{attribute 'linkalways'} 
{attribute 'no_explicit_call' := 'This FB is a CLASS and must be accessed using methods or properties'}
{attribute 'enable_dynamic_creation'}
FUNCTION_BLOCK _TcVnParamsMSER EXTENDS StructuredDatatypeBase
VAR
	localData : TcVnParamsMSER;
	activeData : REFERENCE TO TcVnParamsMSER REF= localData;
	_nDelta : _DINT(localData.nDelta);
    _nMinArea : _UDINT(localData.nMinArea);
	_nMaxArea : _UDINT(localData.nMaxArea);
	_fMaxVariation : _LREAL(localData.fMaxVariation);
	_fMinDiversity : _LREAL(localData.fMinDiversity);
	_nMaxEvolution : _UDINT(localData.nMaxEvolution);
    _fAreaThreshold : _LREAL(localData.fAreaThreshold);
    _fMinMargin : _LREAL(localData.fMinMargin);
    _nEdgeBlurSize : _UDINT(localData.nEdgeBlurSize);
END_VAR

PROPERTY PUBLIC Address : PVOID
GET
Address := ADR(activeData);
END_GET
END_PROPERTY

METHOD PUBLIC ClearReference
VAR_INPUT
END_VAR
activeData REF= localData;
SetMemberReference();
END_METHOD

METHOD PUBLIC Clone : I_Datatype
VAR
    pClone : POINTER TO _TcVnParamsMSER;
END_VAR
pClone := __NEW(_TcVnParamsMSER());
pClone^.Value := Value;
Clone := pClone^;
END_METHOD

PROPERTY PUBLIC fAreaThreshold : REFERENCE TO _LREAL
GET
fAreaThreshold REF= _fAreaThreshold;
END_GET
END_PROPERTY

METHOD FB_init : BOOL
VAR_INPUT
	bInitRetains : BOOL; // if TRUE, the retain variables are initialized (warm start / cold start)
	bInCopyCode : BOOL;  // if TRUE, the instance afterwards gets moved into the copy code (online change)
END_VAR
SetMemberReference();
AddMember('nDelta', _nDelta);
AddMember('nMinArea', _nMinArea);
AddMember('nMaxArea', _nMaxArea);
AddMember('fMaxVariation', _fMaxVariation);
AddMember('fMinDiversity', _fMinDiversity);
AddMember('nMaxEvolution', _nMaxEvolution);
AddMember('fAreaThreshold', _fAreaThreshold);
AddMember('fMinMargin', _fMinMargin);
AddMember('nEdgeBlurSize', _nEdgeBlurSize);
END_METHOD

PROPERTY PUBLIC fMaxVariation : REFERENCE TO _LREAL
GET
fMaxVariation REF= _fMaxVariation;
END_GET
END_PROPERTY

PROPERTY PUBLIC fMinDiversity : REFERENCE TO _LREAL
GET
fMinDiversity REF= _fMinDiversity;
END_GET
END_PROPERTY

PROPERTY PUBLIC fMinMargin : REFERENCE TO _LREAL
GET
fMinMargin REF= _fMinMargin;
END_GET
END_PROPERTY

PROPERTY PUBLIC Identifier : T_MAXSTRING
GET
Identifier := 'TcVnParamsMSER';
END_GET
END_PROPERTY

METHOD PUBLIC MakeReferenceTo
VAR_INPUT
	ReferenceTarget : REFERENCE TO TcVnParamsMSER;
END_VAR
activeData REF= ReferenceTarget;
SetMemberReference();
END_METHOD

PROPERTY PUBLIC nDelta : REFERENCE TO _DINT
GET
nDelta REF= _nDelta;
END_GET
END_PROPERTY

PROPERTY PUBLIC nEdgeBlurSize : REFERENCE TO _UDINT
GET
nEdgeBlurSize REF= _nEdgeBlurSize;
END_GET
END_PROPERTY

PROPERTY PUBLIC nMaxArea : REFERENCE TO _UDINT
GET
nMaxArea REF= _nMaxArea;
END_GET
END_PROPERTY

PROPERTY PUBLIC nMaxEvolution : REFERENCE TO _UDINT
GET
nMaxEvolution REF= _nMaxEvolution;
END_GET
END_PROPERTY

PROPERTY PUBLIC nMinArea : REFERENCE TO _UDINT
GET
nMinArea REF= _nMinArea;
END_GET
END_PROPERTY

METHOD PROTECTED SetMemberReference
VAR_INPUT
END_VAR
_nDelta.MakeReferenceTo(activeData.nDelta);
_nMinArea.MakeReferenceTo(activeData.nMinArea);
_nMaxArea.MakeReferenceTo(activeData.nMaxArea);
_fMaxVariation.MakeReferenceTo(activeData.fMaxVariation);
_fMinDiversity.MakeReferenceTo(activeData.fMinDiversity);
_nMaxEvolution.MakeReferenceTo(activeData.nMaxEvolution);
_fAreaThreshold.MakeReferenceTo(activeData.fAreaThreshold);
_fMinMargin.MakeReferenceTo(activeData.fMinMargin);
_nEdgeBlurSize.MakeReferenceTo(activeData.nEdgeBlurSize);
END_METHOD

PROPERTY PUBLIC Size : UDINT
GET
Size := SIZEOF(activeData);
END_GET
END_PROPERTY

METHOD TryMakeReferenceTo : BOOL
VAR_INPUT
	Target : I_Datatype;
END_VAR
VAR
	pTargetData : POINTER TO TcVnParamsMSER;
END_VAR
IF NOT IsEquivalentTo(Target) THEN
	RETURN;
END_IF

pTargetData := Target.Address;
activeData REF= pTargetData^;
SetMemberReference();
TryMakeReferenceTo := TRUE;
END_METHOD

PROPERTY PUBLIC Value : REFERENCE TO TcVnParamsMSER
GET
Value REF= activeData;
END_GET
END_PROPERTY

END_FUNCTION_BLOCK

(* stored: Version 1.1.0.1, ProductVersion 3.1.4024.13
   POU _TcVnParamsMSER: Id {8415e151-330a-044b-1e44-a5d03d9f1d70}, SpecialFunc None
   Folder Core: Id {0c5e0a5a-b8de-083d-04fa-77bfbde0f7fc}
   Folder Customize: Id {3b0f5d5d-59ec-0949-0a47-6eade71dd329}
   Folder Constructor: Id {73b7aeb2-c2ad-0790-200d-743459cc97ed}
   Folder Protected: Id {f515bbeb-0e88-04dc-3af7-c4b92c5c7383}
   Property Address: Id {15a6aa5f-63a0-069f-3517-43ce737200da}
   Get Get: Id {9157615d-2420-03f3-131a-2fd2e7a7b131}
   Method ClearReference: Id {619a585a-5063-0959-02ce-050b17f19f79}
   Method Clone: Id {c85bec7d-5e4e-0d5c-191a-28926f3375d0}
   Property fAreaThreshold: Id {5dfb13a4-7ba9-05fd-0a18-bf3f8b5c0d1a}
   Get Get: Id {9ae9a7fa-acf3-096c-0edb-1531b715af56}
   Method FB_init: Id {17de168b-30c3-00fb-29e7-e10e1259deb0}
   Property fMaxVariation: Id {1c3f244e-6610-0f65-1409-0cd93a8a074e}
   Get Get: Id {4229a383-bcc7-07f6-21b6-5923286ac9fa}
   Property fMinDiversity: Id {de617d27-07d6-018e-18c3-eec4738b986d}
   Get Get: Id {801d4649-10a4-0c36-26e9-e57c0668b74e}
   Property fMinMargin: Id {b8c5977f-1109-0c74-0143-f78ca74926ff}
   Get Get: Id {6f59f1ea-56c5-032b-1b59-eec8fd4fe09a}
   Property Identifier: Id {9db0f63e-fd08-0682-308e-966c5b16313b}
   Get Get: Id {a28e4e79-2a55-08dd-2477-1915f3c3af09}
   Method MakeReferenceTo: Id {4f5a33b5-30cc-01aa-2b27-9ee9dd8f386a}
   Property nDelta: Id {90823a2d-b3f3-03b6-3ee6-f0de1daf1716}
   Get Get: Id {a4489dac-7411-0301-362f-4bd46ec5b088}
   Property nEdgeBlurSize: Id {8a082ef8-77f7-07eb-26a6-0a95a3875a37}
   Get Get: Id {17e6ed4a-9ceb-0fc4-0865-8eb3af4b170c}
   Property nMaxArea: Id {99d875f8-e939-04b5-0bb6-b2fcd5a96b16}
   Get Get: Id {6f5ea55b-00e2-03c7-32ef-01d3d48e1ad5}
   Property nMaxEvolution: Id {c7f6463d-bdfc-00e0-367c-2360bc7733b2}
   Get Get: Id {8dff4dde-2540-064e-1562-a4f9f4fe9a3f}
   Property nMinArea: Id {950b61eb-cad8-0a2f-1acd-51fee0ddf165}
   Get Get: Id {6dda2a1b-1a23-01dc-2d7f-11425cbd6d85}
   Method SetMemberReference: Id {37de610e-3f62-09c2-3a20-7f2bf78f6329}
   Property Size: Id {a065791b-fa96-0998-0229-e77b3362b3ff}
   Get Get: Id {9bf6a221-d182-0202-321e-90a6731fe711}
   Method TryMakeReferenceTo: Id {bc392d66-6ef0-0b57-03dc-a166add914c7}
   Property Value: Id {10f951fb-2b6e-089a-1ae8-7e36ccad7693}
   Get Get: Id {a52f3280-a601-06d7-3d3a-aa4877ae2990} *)
